TYPE ST_ProductStats :
STRUCT
	 averageWeight : REAL;
     minWeight     : REAL;
	 maxWeight     : REAL;
	 defectiveCount: INT;
END_STRUCT
END_TYPE

(* stored: Version 1.1.0.1, ProductVersion 3.1.4024.16
   DUT ST_ProductStats: Id {a513677f-6ce6-4794-ae9e-3ddc35f1d31a} *)
